// Mitsubishi GX Works2 project: exam_practice   PLC: Q02/Q02H

PROGRAM Q5-MC
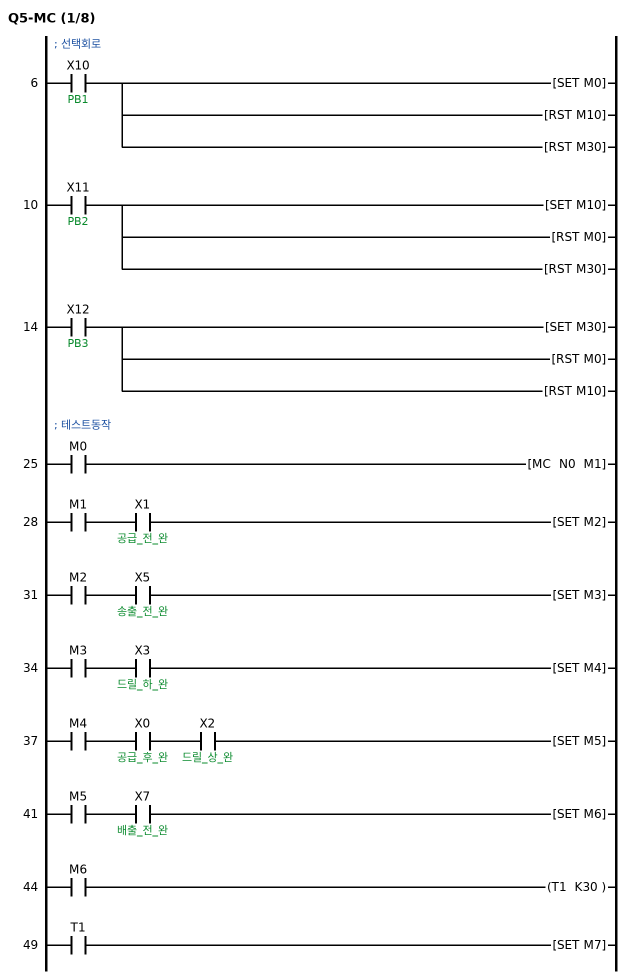
; 선택회로
6     LD      X10  ; PB1
      SET     M0
      RST     M10
      RST     M30
10    LD      X11  ; PB2
      SET     M10
      RST     M0
      RST     M30
14    LD      X12  ; PB3
      SET     M30
      RST     M0
      RST     M10
; 테스트동작
25    LD      M0
      MC      N0 M1
28    LD      M1
      AND     X1  ; 공급_전_완
      SET     M2
31    LD      M2
      AND     X5  ; 송출_전_완
      SET     M3
34    LD      M3
      AND     X3  ; 드릴_하_완
      SET     M4
37    LD      M4
      AND     X0  ; 공급_후_완
      AND     X2  ; 드릴_상_완
      SET     M5
41    LD      M5
      AND     X7  ; 배출_전_완
      SET     M6
44    LD      M6
      OUT     T1 K30
49    LD      T1
      SET     M7
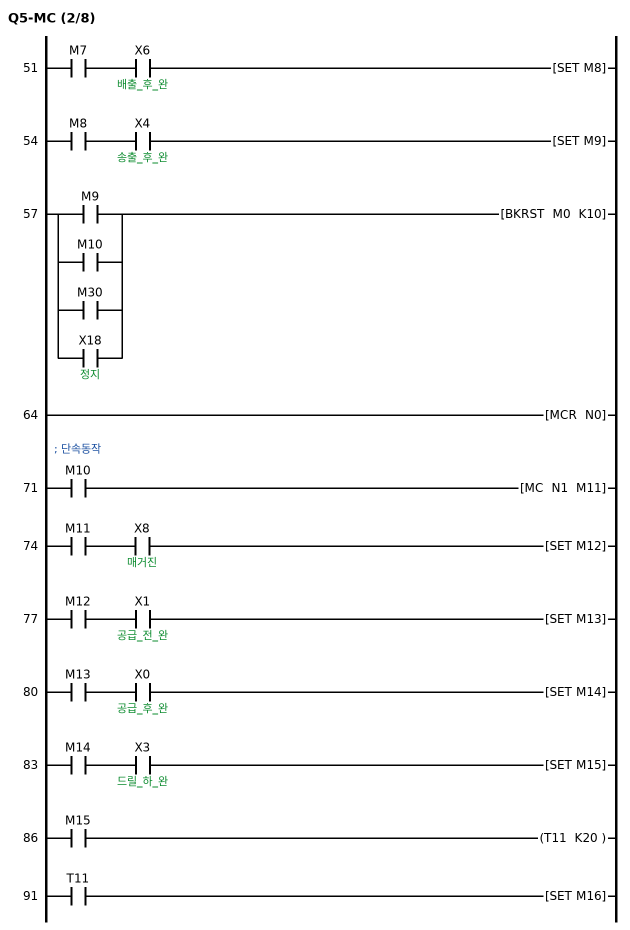
51    LD      M7
      AND     X6  ; 배출_후_완
      SET     M8
54    LD      M8
      AND     X4  ; 송출_후_완
      SET     M9
57    LD      M9
      OR      M10
      OR      M30
      OR      X18  ; 정지
      BKRST   M0 K10
64    MCR     N0
; 단속동작
71    LD      M10
      MC      N1 M11
74    LD      M11
      AND     X8  ; 매거진
      SET     M12
77    LD      M12
      AND     X1  ; 공급_전_완
      SET     M13
80    LD      M13
      AND     X0  ; 공급_후_완
      SET     M14
83    LD      M14
      AND     X3  ; 드릴_하_완
      SET     M15
86    LD      M15
      OUT     T11 K20
91    LD      T11
      SET     M16
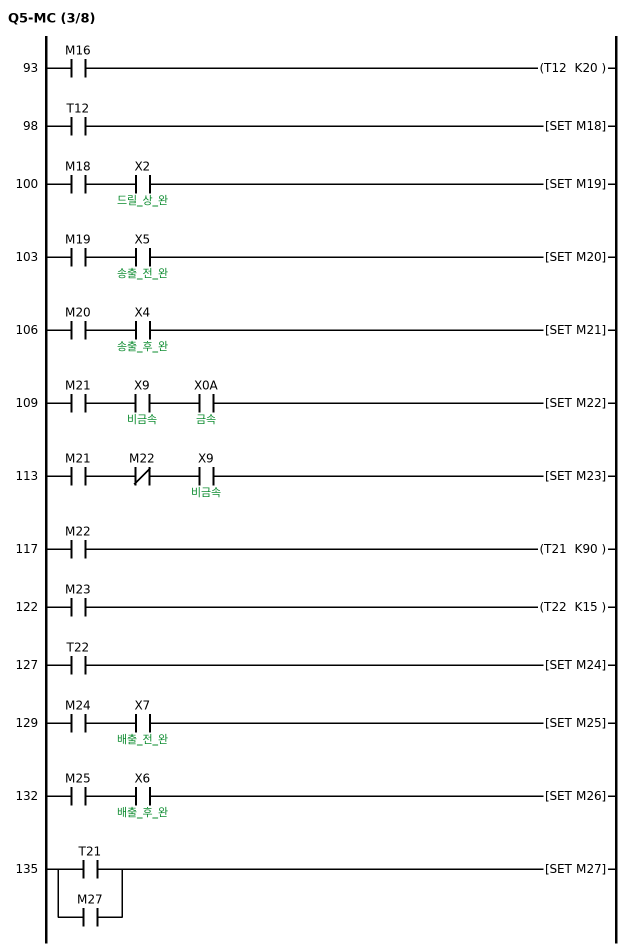
93    LD      M16
      OUT     T12 K20
98    LD      T12
      SET     M18
100   LD      M18
      AND     X2  ; 드릴_상_완
      SET     M19
103   LD      M19
      AND     X5  ; 송출_전_완
      SET     M20
106   LD      M20
      AND     X4  ; 송출_후_완
      SET     M21
109   LD      M21
      AND     X9  ; 비금속
      AND     X0A  ; 금속
      SET     M22
113   LD      M21
      ANI     M22
      AND     X9  ; 비금속
      SET     M23
117   LD      M22
      OUT     T21 K90
122   LD      M23
      OUT     T22 K15
127   LD      T22
      SET     M24
129   LD      M24
      AND     X7  ; 배출_전_완
      SET     M25
132   LD      M25
      AND     X6  ; 배출_후_완
      SET     M26
135   LD      T21
      OR      M27
      SET     M27
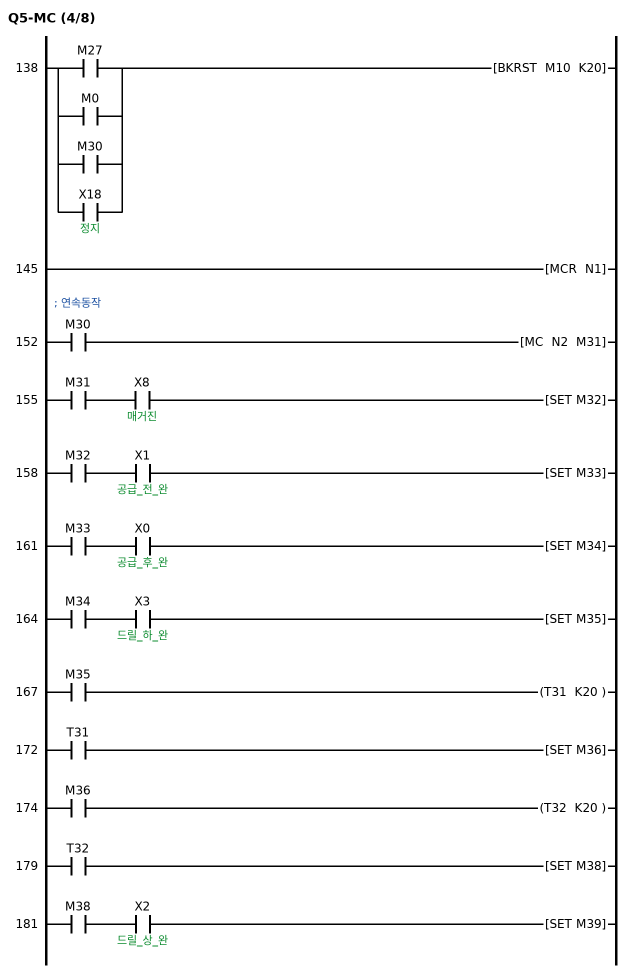
138   LD      M27
      OR      M0
      OR      M30
      OR      X18  ; 정지
      BKRST   M10 K20
145   MCR     N1
; 연속동작
152   LD      M30
      MC      N2 M31
155   LD      M31
      AND     X8  ; 매거진
      SET     M32
158   LD      M32
      AND     X1  ; 공급_전_완
      SET     M33
161   LD      M33
      AND     X0  ; 공급_후_완
      SET     M34
164   LD      M34
      AND     X3  ; 드릴_하_완
      SET     M35
167   LD      M35
      OUT     T31 K20
172   LD      T31
      SET     M36
174   LD      M36
      OUT     T32 K20
179   LD      T32
      SET     M38
181   LD      M38
      AND     X2  ; 드릴_상_완
      SET     M39
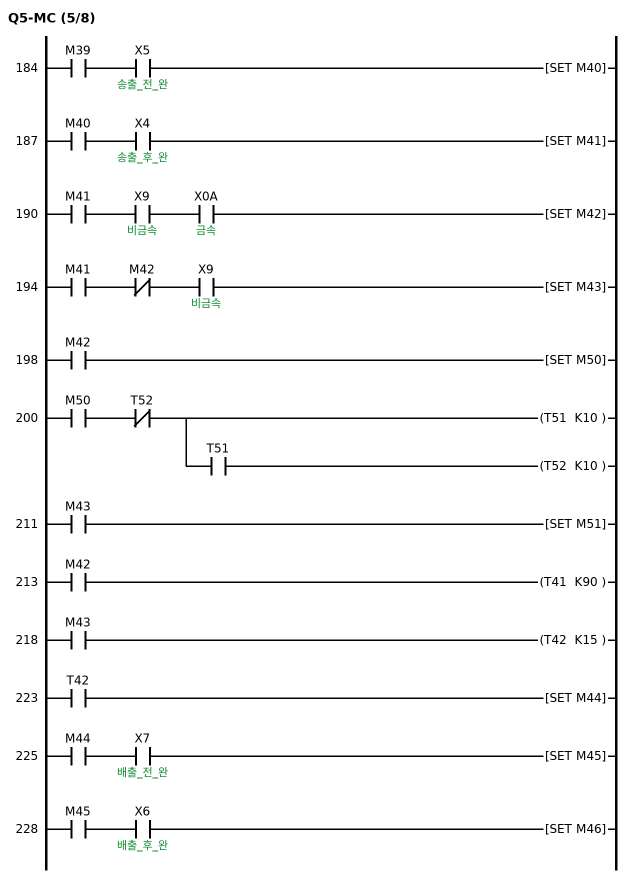
184   LD      M39
      AND     X5  ; 송출_전_완
      SET     M40
187   LD      M40
      AND     X4  ; 송출_후_완
      SET     M41
190   LD      M41
      AND     X9  ; 비금속
      AND     X0A  ; 금속
      SET     M42
194   LD      M41
      ANI     M42
      AND     X9  ; 비금속
      SET     M43
198   LD      M42
      SET     M50
200   LD      M50
      ANI     T52
      OUT     T51 K10
      AND     T51
      OUT     T52 K10
211   LD      M43
      SET     M51
213   LD      M42
      OUT     T41 K90
218   LD      M43
      OUT     T42 K15
223   LD      T42
      SET     M44
225   LD      M44
      AND     X7  ; 배출_전_완
      SET     M45
228   LD      M45
      AND     X6  ; 배출_후_완
      SET     M46
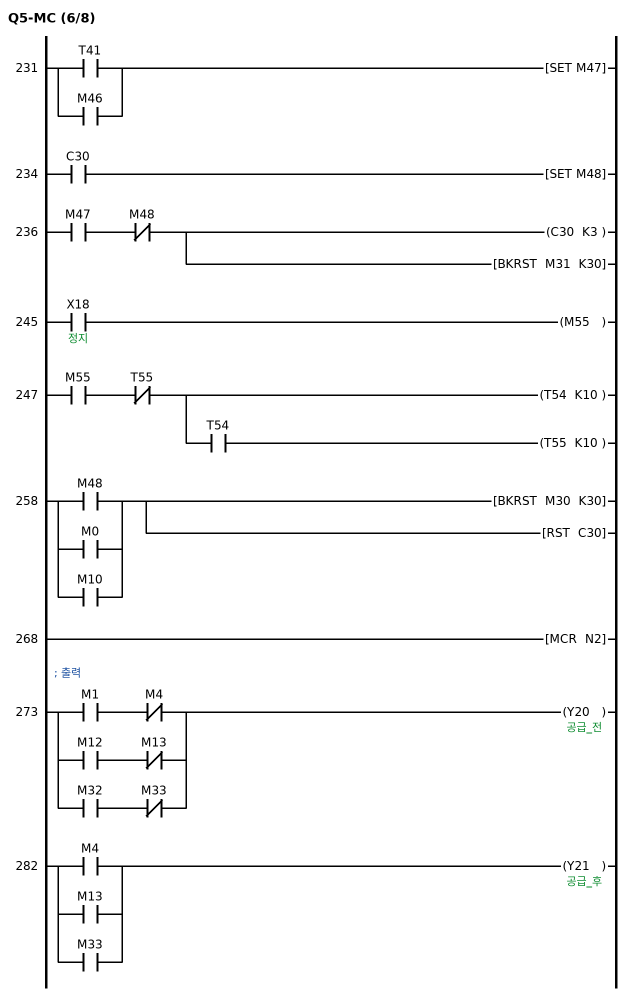
231   LD      T41
      OR      M46
      SET     M47
234   LD      C30
      SET     M48
236   LD      M47
      ANI     M48
      OUT     C30 K3
      BKRST   M31 K30
245   LD      X18  ; 정지
      OUT     M55
247   LD      M55
      ANI     T55
      OUT     T54 K10
      AND     T54
      OUT     T55 K10
258   LD      M48
      OR      M0
      OR      M10
      BKRST   M30 K30
      RST     C30
268   MCR     N2
; 출력
273   LD      M1
      ANI     M4
      LD      M12
      ANI     M13
      ORB
      LD      M32
      ANI     M33
      ORB
      OUT     Y20  ; 공급_전
282   LD      M4
      OR      M13
      OR      M33
      OUT     Y21  ; 공급_후
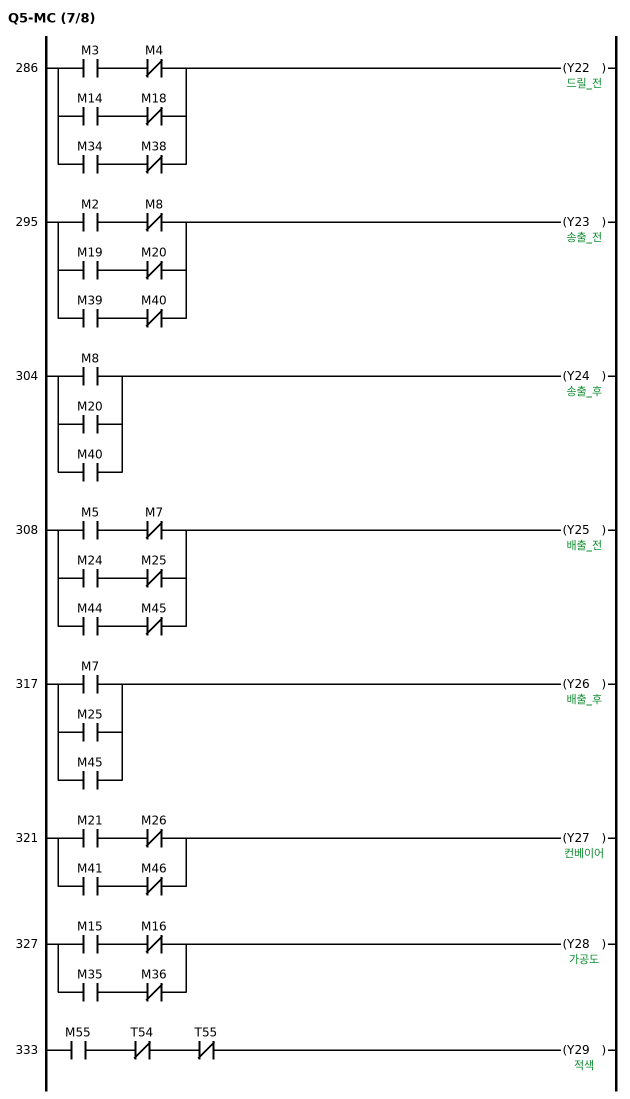
286   LD      M3
      ANI     M4
      LD      M14
      ANI     M18
      ORB
      LD      M34
      ANI     M38
      ORB
      OUT     Y22  ; 드릴_전
295   LD      M2
      ANI     M8
      LD      M19
      ANI     M20
      ORB
      LD      M39
      ANI     M40
      ORB
      OUT     Y23  ; 송출_전
304   LD      M8
      OR      M20
      OR      M40
      OUT     Y24  ; 송출_후
308   LD      M5
      ANI     M7
      LD      M24
      ANI     M25
      ORB
      LD      M44
      ANI     M45
      ORB
      OUT     Y25  ; 배출_전
317   LD      M7
      OR      M25
      OR      M45
      OUT     Y26  ; 배출_후
321   LD      M21
      ANI     M26
      LD      M41
      ANI     M46
      ORB
      OUT     Y27  ; 컨베이어
327   LD      M15
      ANI     M16
      LD      M35
      ANI     M36
      ORB
      OUT     Y28  ; 가공도
333   LD      M55
      ANI     T54
      ANI     T55
      OUT     Y29  ; 적색
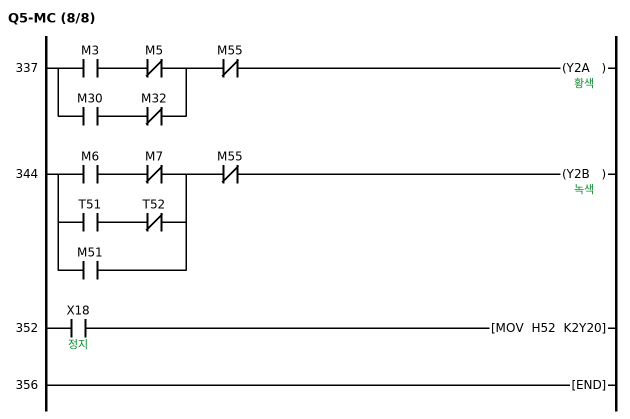
337   LD      M3
      ANI     M5
      LD      M30
      ANI     M32
      ORB
      ANI     M55
      OUT     Y2A  ; 황색
344   LD      M6
      ANI     M7
      LD      T51
      ANI     T52
      ORB
      OR      M51
      ANI     M55
      OUT     Y2B  ; 녹색
352   LD      X18  ; 정지
      MOV     H52 K2Y20
356   END
END_PROGRAM

PROGRAM exam_q9
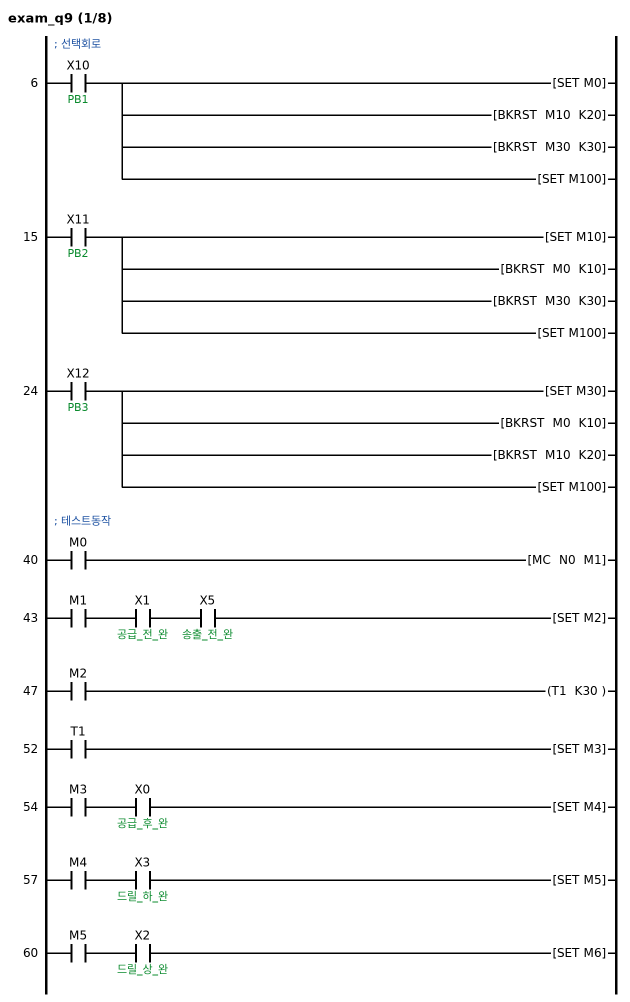
; 선택회로
6     LD      X10  ; PB1
      SET     M0
      BKRST   M10 K20
      BKRST   M30 K30
      SET     M100
15    LD      X11  ; PB2
      SET     M10
      BKRST   M0 K10
      BKRST   M30 K30
      SET     M100
24    LD      X12  ; PB3
      SET     M30
      BKRST   M0 K10
      BKRST   M10 K20
      SET     M100
; 테스트동작
40    LD      M0
      MC      N0 M1
43    LD      M1
      AND     X1  ; 공급_전_완
      AND     X5  ; 송출_전_완
      SET     M2
47    LD      M2
      OUT     T1 K30
52    LD      T1
      SET     M3
54    LD      M3
      AND     X0  ; 공급_후_완
      SET     M4
57    LD      M4
      AND     X3  ; 드릴_하_완
      SET     M5
60    LD      M5
      AND     X2  ; 드릴_상_완
      SET     M6
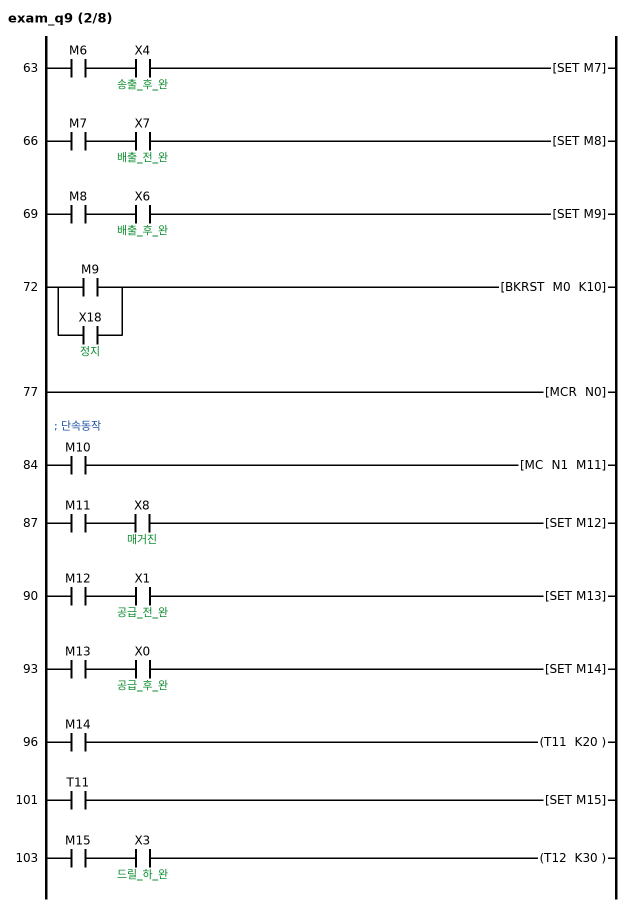
63    LD      M6
      AND     X4  ; 송출_후_완
      SET     M7
66    LD      M7
      AND     X7  ; 배출_전_완
      SET     M8
69    LD      M8
      AND     X6  ; 배출_후_완
      SET     M9
72    LD      M9
      OR      X18  ; 정지
      BKRST   M0 K10
77    MCR     N0
; 단속동작
84    LD      M10
      MC      N1 M11
87    LD      M11
      AND     X8  ; 매거진
      SET     M12
90    LD      M12
      AND     X1  ; 공급_전_완
      SET     M13
93    LD      M13
      AND     X0  ; 공급_후_완
      SET     M14
96    LD      M14
      OUT     T11 K20
101   LD      T11
      SET     M15
103   LD      M15
      AND     X3  ; 드릴_하_완
      OUT     T12 K30
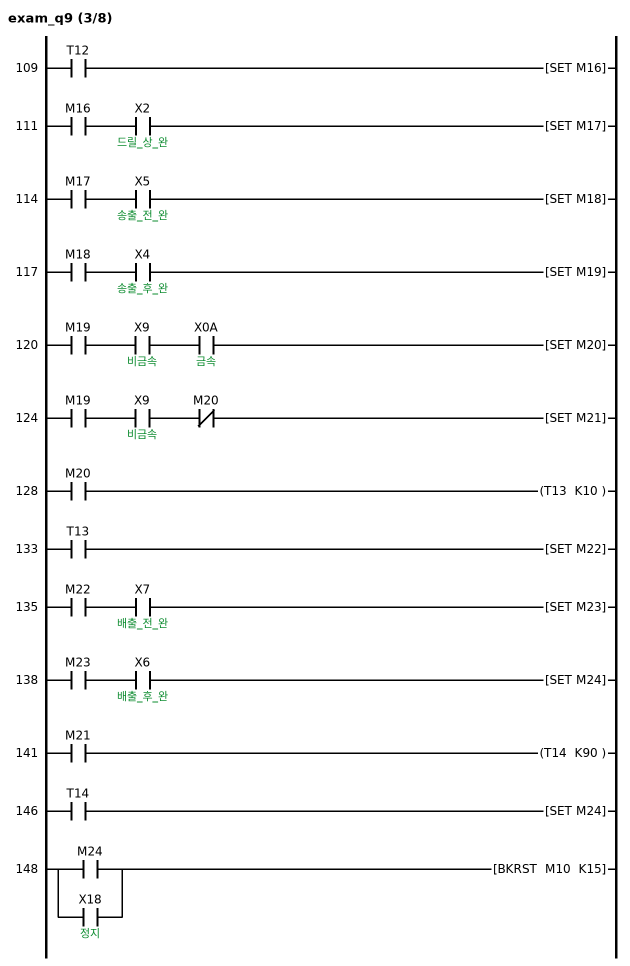
109   LD      T12
      SET     M16
111   LD      M16
      AND     X2  ; 드릴_상_완
      SET     M17
114   LD      M17
      AND     X5  ; 송출_전_완
      SET     M18
117   LD      M18
      AND     X4  ; 송출_후_완
      SET     M19
120   LD      M19
      AND     X9  ; 비금속
      AND     X0A  ; 금속
      SET     M20
124   LD      M19
      AND     X9  ; 비금속
      ANI     M20
      SET     M21
128   LD      M20
      OUT     T13 K10
133   LD      T13
      SET     M22
135   LD      M22
      AND     X7  ; 배출_전_완
      SET     M23
138   LD      M23
      AND     X6  ; 배출_후_완
      SET     M24
141   LD      M21
      OUT     T14 K90
146   LD      T14
      SET     M24
148   LD      M24
      OR      X18  ; 정지
      BKRST   M10 K15
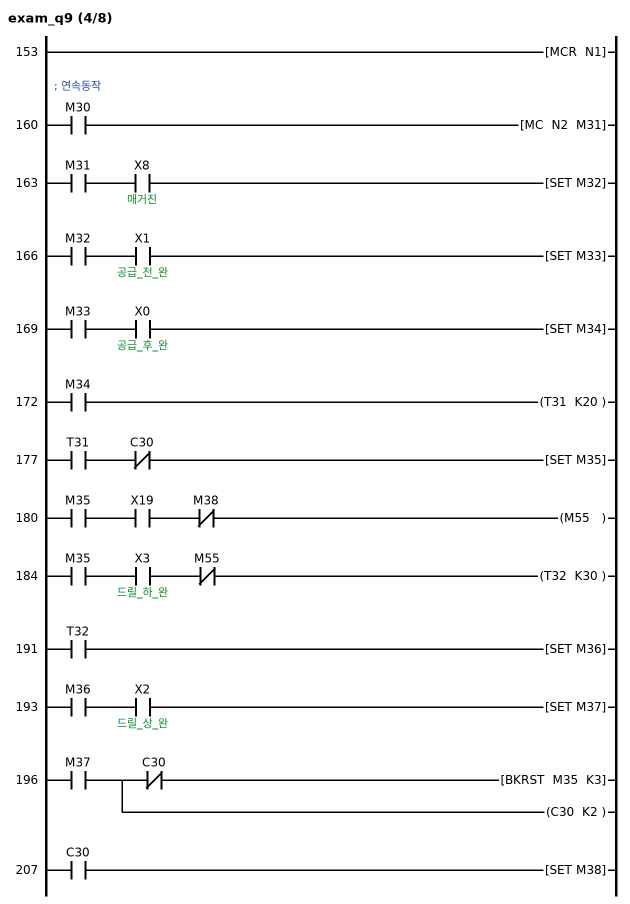
153   MCR     N1
; 연속동작
160   LD      M30
      MC      N2 M31
163   LD      M31
      AND     X8  ; 매거진
      SET     M32
166   LD      M32
      AND     X1  ; 공급_전_완
      SET     M33
169   LD      M33
      AND     X0  ; 공급_후_완
      SET     M34
172   LD      M34
      OUT     T31 K20
177   LD      T31
      ANI     C30
      SET     M35
180   LD      M35
      AND     X19
      ANI     M38
      OUT     M55
184   LD      M35
      AND     X3  ; 드릴_하_완
      ANI     M55
      OUT     T32 K30
191   LD      T32
      SET     M36
193   LD      M36
      AND     X2  ; 드릴_상_완
      SET     M37
196   LD      M37
      MPS
      ANI     C30
      BKRST   M35 K3
      MPP
      OUT     C30 K2
207   LD      C30
      SET     M38
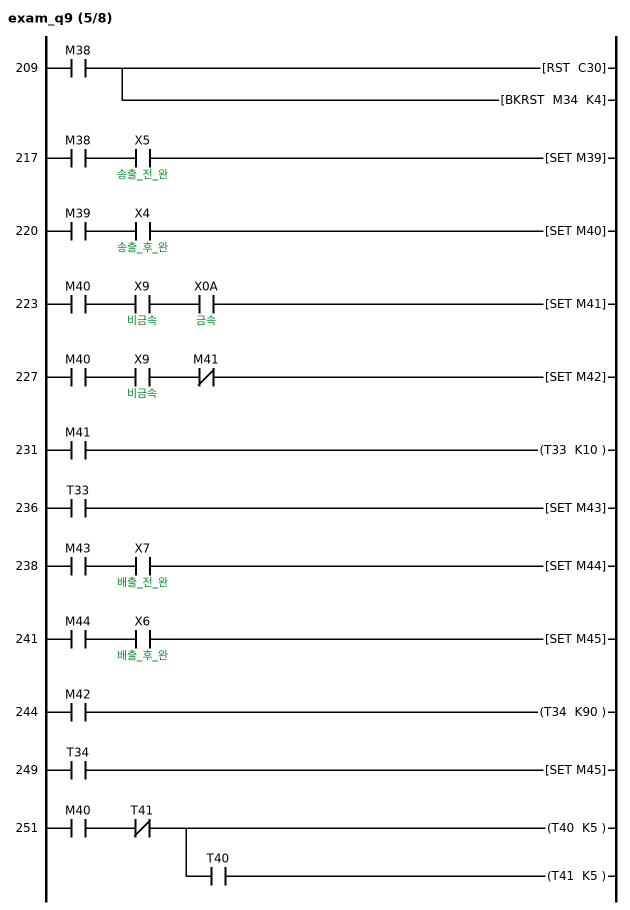
209   LD      M38
      RST     C30
      BKRST   M34 K4
217   LD      M38
      AND     X5  ; 송출_전_완
      SET     M39
220   LD      M39
      AND     X4  ; 송출_후_완
      SET     M40
223   LD      M40
      AND     X9  ; 비금속
      AND     X0A  ; 금속
      SET     M41
227   LD      M40
      AND     X9  ; 비금속
      ANI     M41
      SET     M42
231   LD      M41
      OUT     T33 K10
236   LD      T33
      SET     M43
238   LD      M43
      AND     X7  ; 배출_전_완
      SET     M44
241   LD      M44
      AND     X6  ; 배출_후_완
      SET     M45
244   LD      M42
      OUT     T34 K90
249   LD      T34
      SET     M45
251   LD      M40
      ANI     T41
      OUT     T40 K5
      AND     T40
      OUT     T41 K5
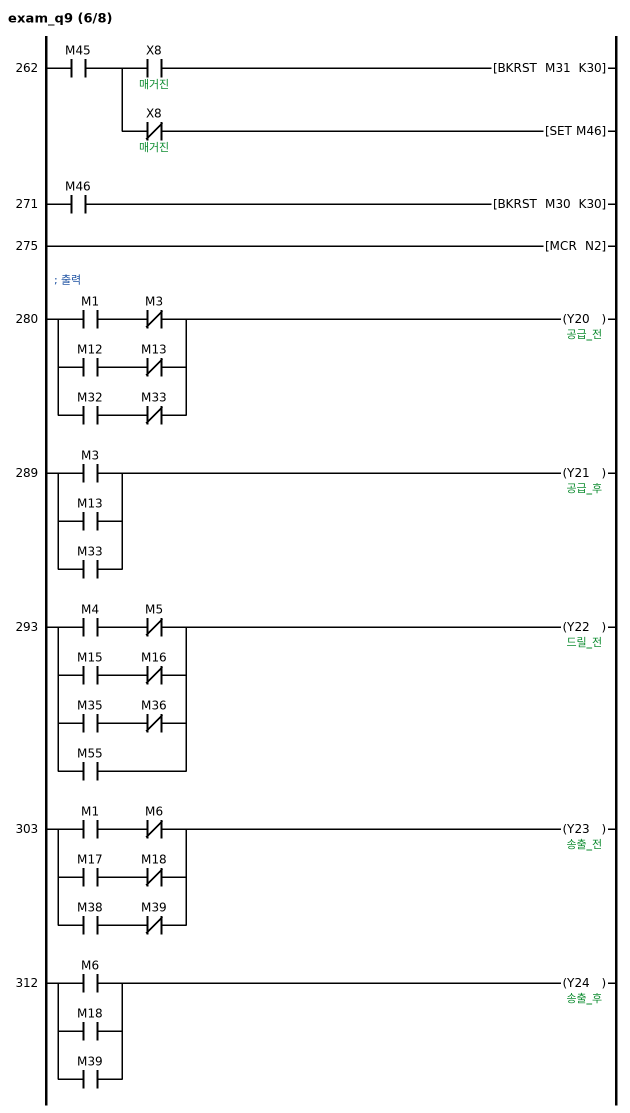
262   LD      M45
      MPS
      AND     X8  ; 매거진
      BKRST   M31 K30
      MPP
      ANI     X8  ; 매거진
      SET     M46
271   LD      M46
      BKRST   M30 K30
275   MCR     N2
; 출력
280   LD      M1
      ANI     M3
      LD      M12
      ANI     M13
      ORB
      LD      M32
      ANI     M33
      ORB
      OUT     Y20  ; 공급_전
289   LD      M3
      OR      M13
      OR      M33
      OUT     Y21  ; 공급_후
293   LD      M4
      ANI     M5
      LD      M15
      ANI     M16
      ORB
      LD      M35
      ANI     M36
      ORB
      OR      M55
      OUT     Y22  ; 드릴_전
303   LD      M1
      ANI     M6
      LD      M17
      ANI     M18
      ORB
      LD      M38
      ANI     M39
      ORB
      OUT     Y23  ; 송출_전
312   LD      M6
      OR      M18
      OR      M39
      OUT     Y24  ; 송출_후
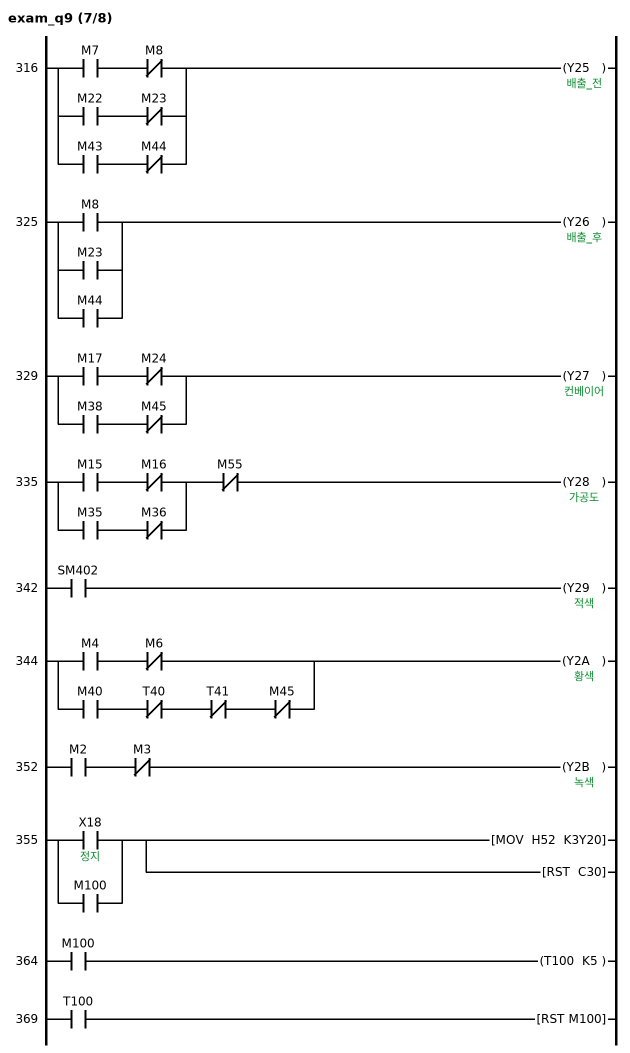
316   LD      M7
      ANI     M8
      LD      M22
      ANI     M23
      ORB
      LD      M43
      ANI     M44
      ORB
      OUT     Y25  ; 배출_전
325   LD      M8
      OR      M23
      OR      M44
      OUT     Y26  ; 배출_후
329   LD      M17
      ANI     M24
      LD      M38
      ANI     M45
      ORB
      OUT     Y27  ; 컨베이어
335   LD      M15
      ANI     M16
      LD      M35
      ANI     M36
      ORB
      ANI     M55
      OUT     Y28  ; 가공도
342   LD      SM402
      OUT     Y29  ; 적색
344   LD      M4
      ANI     M6
      LD      M40
      ANI     T40
      ANI     T41
      ANI     M45
      ORB
      OUT     Y2A  ; 황색
352   LD      M2
      ANI     M3
      OUT     Y2B  ; 녹색
355   LD      X18  ; 정지
      OR      M100
      MOV     H52 K3Y20
      RST     C30
364   LD      M100
      OUT     T100 K5
369   LD      T100
      RST     M100
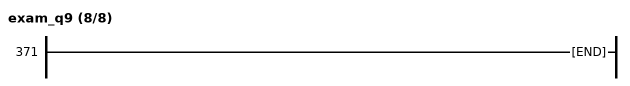
371   END
END_PROGRAM
